Yaskawa INFORM job: OK_R2_O38-47,64(2)(90,0)_MPOK.JBI

/JOB
//NAME OK_R2_O38-47,64(2)(90,0)_MPOK
///FOLDERNAME X4
//POS
///NPOS 359,359,359,19,0,0
///TOOL 0
///POSTYPE PULSE
///PULSE
C00000=-102904,-190754,-108658,-56793,33718,43054
C00001=-112112,-124440,-79629,-37912,40591,30924
C00002=-145621,-43895,-45824,-14341,74181,8322
C00003=-153971,-33006,-36006,-12070,72386,5523
C00004=-154957,-31241,-33389,-11833,71552,5253
C00005=-154957,-31059,-32306,-11871,70990,5309
C00006=-154957,-31147,-32820,-11853,71255,5283
C00007=-152959,-34045,-35008,-12435,71415,5986
C00008=-152821,-33501,-33767,-12507,70963,6084
C00009=-152893,-32341,-33000,-12478,71072,6047
C00010=-153154,-34489,-35846,-12359,71666,5891
C00011=-152546,-38024,-38116,-12561,71351,6144
C00012=-150032,-44426,-43245,-13273,71622,7027
C00013=-145621,-43895,-45824,-14341,74181,8322
C00014=-126188,-124725,-79701,-29915,35046,24780
C00015=-102904,-190754,-108658,-56793,33718,43054
C00016=-131529,-189509,-110128,-36771,24434,27261
C00017=-124211,-86804,-80218,-19393,77786,15538
C00018=-160160,17664,-548,-10057,75687,3034
C00019=-160660,22954,7322,-10002,73531,3037
C00020=-166212,32109,17444,-8387,71396,1231
C00021=-166212,32264,18572,-8416,70786,1274
C00022=-166212,32192,18060,-8403,71061,1255
C00023=-166132,29456,15334,-8416,71338,1265
C00024=-166132,29543,15979,-8433,70989,1289
C00025=-166315,30482,16900,-8379,70890,1229
C00026=-166283,28892,15324,-8381,71043,1230
C00027=-165319,19573,3695,-8574,73487,1399
C00028=-163582,7043,-11027,-8999,76267,1804
C00029=-162101,-9402,-41897,-5301,86162,910
C00030=-133469,39121,-1061,931,85072,6891
C00031=-135751,46408,8355,1655,83056,6142
C00032=-135516,49476,14058,1587,81119,6193
C00033=-135516,49311,14679,1588,80652,6188
C00034=-135036,46950,11602,1434,81323,6352
C00035=-134946,46723,11962,1405,80982,6377
C00036=-135074,47950,13285,1445,80801,6333
C00037=-135102,44394,8734,1452,81774,6335
C00038=-133469,39121,-1061,931,85072,6891
C00039=-135146,16919,-22910,1456,87131,6386
C00040=-160578,-137207,-111137,27103,45167,-7155
C00041=-166532,-153428,-115250,33739,42272,-11545
C00042=-166532,-153428,-115250,33739,42272,-11545
C00043=-160883,-131526,-133102,-3483,78120,-6366
C00044=-103370,-159686,-136025,-1765,64172,-8056
C00045=-97179,-138237,-129333,-10238,76593,11306
C00046=-96065,-128281,-122439,-10507,77596,11607
C00047=-96065,-128106,-120653,-10546,76604,11690
C00048=-96065,-128281,-122439,-10507,77596,11607
C00049=-96974,-121186,-120234,-10189,79734,11117
C00050=-96065,-128281,-122439,-10507,77596,11607
C00051=-80019,-98046,-111669,-14399,88698,15911
C00052=-80077,-97852,-111516,-14385,88694,15892
C00053=-80077,-98331,-110658,-14385,87944,15982
C00054=-80077,-97897,-111441,-14385,88627,15900
C00055=-80867,-94680,-110202,-14197,89359,15553
C00056=-80077,-97897,-111441,-14385,88627,15900
C00057=-77060,-103837,-123440,-15157,93336,16325
C00058=-77104,-103620,-123385,-15148,93404,16303
C00059=-82212,-117279,-126602,-8714,87753,18646
C00060=-83304,-119533,-127995,-7425,87342,19011
C00061=-83304,-120285,-126924,-7427,86307,19072
C00062=-83304,-120125,-127175,-7427,86540,19060
C00063=-84285,-114583,-125380,-7184,88184,18645
C00064=-83304,-120125,-127175,-7427,86540,19060
C00065=-78124,-131037,-133000,-8681,85036,20864
C00066=-78124,-131037,-133000,-8681,85036,20864
C00067=-80781,-132367,-131851,-8063,83392,20088
C00068=-80781,-132658,-130737,-8071,82565,20142
C00069=-80781,-132579,-131090,-8068,82820,20125
C00070=-82215,-124520,-128659,-7695,85306,19491
C00071=-80136,-136061,-133167,-8229,82377,20371
C00072=-80218,-134686,-135534,-8183,84509,20204
C00073=-75563,-118157,-129697,-13391,92336,27261
C00074=-84024,-123631,-127734,-11595,87159,24981
C00075=-84024,-123979,-126960,-11598,86516,25042
C00076=-84024,-123746,-127494,-11596,86956,25000
C00077=-85048,-122093,-126977,-11373,87337,24623
C00078=-81994,-135324,-132084,-12059,84184,25946
C00079=-81994,-133752,-136174,-12028,87438,25630
C00080=-81994,-133752,-136174,-12028,87438,25630
C00081=-83107,-120864,-125937,-11789,87596,25245
C00082=-83880,-119254,-122492,-11630,86222,25116
C00083=-83880,-119583,-121326,-11637,85351,25197
C00084=-83880,-119399,-122020,-11633,85865,25149
C00085=-85062,-113328,-120022,-11369,87556,24598
C00086=-83880,-119399,-122020,-11633,85865,25149
C00087=-83464,-119333,-123502,-11716,86850,25194
C00088=-84085,-116294,-122008,-11580,87393,24935
C00089=-84085,-116863,-120480,-11583,86184,25047
C00090=-84085,-116689,-121008,-11580,86590,25010
C00091=-85140,-111307,-119205,-11348,88071,24523
C00092=-84085,-116194,-122230,-11576,87577,24918
C00093=-82864,-118268,-130611,-11862,91757,24924
C00094=-82864,-118268,-130611,-11862,91757,24924
C00095=-86851,-110557,-120071,-10968,88745,23893
C00096=-86851,-111341,-118540,-10968,87421,24011
C00097=-86851,-110811,-119621,-10968,88345,23929
C00098=-88598,-109546,-119189,-10575,88500,23337
C00099=-86851,-110811,-119621,-10968,88345,23929
C00100=-83825,-124590,-131318,-11630,88867,24881
C00101=-82909,-127853,-136097,-11834,90233,25054
C00102=-84148,-125178,-125504,-11579,85018,25131
C00103=-81186,-118241,-121828,-12198,86718,25964
C00104=-81186,-118533,-120824,-12201,85966,26037
C00105=-81186,-118483,-121017,-12200,86107,26023
C00106=-82314,-113243,-119285,-11952,87535,25506
C00107=-81186,-118241,-121828,-12198,86718,25964
C00108=-87931,-140644,-131144,-10841,80108,24284
C00109=-89960,-139833,-128047,-10433,78377,23732
C00110=-89960,-139550,-127065,-10448,77925,23770
C00111=-89960,-139622,-127307,-10444,78035,23761
C00112=-90753,-134395,-125809,-10209,79670,23349
C00113=-89456,-143397,-129529,-10578,77538,23979
C00114=-95203,-107502,-133483,-6717,98684,21003
C00115=-95203,-107502,-133483,-6717,98684,21003
C00116=70091,-137861,-134613,19540,89589,-11549
C00117=70091,-137861,-134613,19540,89589,-11549
C00118=89914,-142582,-130695,14485,81723,-10120
C00119=90202,-137048,-128128,14398,82897,-9883
C00120=90202,-136718,-126391,14423,82025,-9985
C00121=90202,-136862,-127082,14413,82365,-9945
C00122=91010,-131454,-125503,14223,83978,-9478
C00123=90202,-137070,-128271,14397,82970,-9874
C00124=76195,-137070,-128271,14397,82970,-9874
C00125=74994,-123934,-123423,14560,86840,-9835
C00126=74994,-124092,-122198,14564,86029,-9931
C00127=74994,-124005,-122955,14561,86525,-9872
C00128=76141,-119465,-121513,14342,87728,-9340
C00129=72631,-133219,-128550,14998,85696,-10781
C00130=72631,-131663,-134232,14989,89852,-10278
C00131=50716,-132590,-134806,14983,95067,-21778
C00132=53786,-122460,-125023,14607,93736,-20890
C00133=54881,-121663,-124068,14472,93371,-20558
C00134=54881,-122014,-122728,14450,92397,-20672
C00135=54881,-121856,-123398,14460,92875,-20616
C00136=56721,-117465,-121986,14267,93906,-19868
C00137=54881,-121856,-123398,14460,92875,-20616
C00138=55322,-120745,-123309,14420,93300,-20415
C00139=55322,-120747,-123302,14420,93295,-20416
C00140=55322,-120978,-122461,14407,92679,-20487
C00141=55322,-120864,-122902,14414,92999,-20450
C00142=56710,-117554,-121835,14266,93775,-19889
C00143=54436,-122887,-123768,14509,92662,-20793
C00144=54436,-122067,-126198,14556,94519,-20574
C00145=53688,-126302,-127242,14482,93230,-21000
C00146=7968,-117738,-135568,14910,102458,-19890
C00147=7968,-117738,-135568,14910,102458,-19890
C00148=4119,-116606,-125698,15061,97809,-21757
C00149=7770,-114903,-122318,14590,96007,-20739
C00150=7770,-115418,-121244,14557,95111,-20843
C00151=7770,-115024,-122084,14598,95810,-20761
C00152=9375,-110655,-120613,14452,96836,-20097
C00153=7770,-115024,-122084,14598,95810,-20761
C00154=10569,-102485,-118509,17167,107955,-30726
C00155=17008,-101176,-116544,17116,107524,-30934
C00156=-121481,-92648,-105286,-5369,115019,-86755
C00157=-120615,-96829,-107734,-5213,114434,-86412
C00158=23859,-150611,-131722,11614,81196,-13147
C00159=5605,-98558,-114313,9016,91646,-19053
C00160=5292,-97369,-113802,9089,91971,-19129
C00161=5881,-109040,-123705,8960,92007,-18939
C00162=6434,-120006,-133010,8839,92040,-18760
C00163=-12667,-120051,-129788,-19636,91452,63850
C00164=-15640,-171133,-136982,-20070,70138,66271
C00165=3779,-163113,-125940,-36463,74354,73480
C00166=-120436,-95190,-80290,-14692,43277,16053
C00167=-119715,-95468,-78930,-15521,42464,16563
C00168=1349,-140937,-118482,-38247,78517,71026
C00169=-15636,-141614,-117585,-35447,65083,67762
C00170=-17609,-126505,-112505,-34601,67163,66072
C00171=-24043,-118481,-124771,-21586,79008,61529
C00172=-24043,-118481,-124771,-21586,79008,61529
C00173=-75030,-118005,-124618,-21594,79160,61521
C00174=-115715,-153549,-128562,15788,54400,49074
C00175=-122131,-153692,-122292,24372,49463,44977
C00176=-120438,-96789,-101713,-1489,48968,3516
C00177=-120356,-99154,-104149,-1548,49253,3547
C00178=-84198,-116806,-111213,1772,54897,61304
C00179=-87160,-120534,-109364,10018,48087,58269
C00180=-90828,-138253,-118809,13315,45388,56216
C00181=-90828,-138253,-118809,13315,45388,56216
C00182=-90828,-142934,-129815,12421,49655,56806
C00183=-90829,-142933,-129813,12421,49658,56806
C00184=-119872,-163920,-132846,33283,49576,42941
C00185=-126991,-146326,-124104,35016,55490,41598
C00186=-120835,-94912,-106201,4597,84031,3620
C00187=-120296,-100536,-106811,4468,81494,3706
C00188=-119922,-143587,-123205,31413,53438,44308
C00189=-77415,-98459,-105381,5383,51560,63214
C00190=-71925,-92447,-101662,533,50488,65336
C00191=-77718,-122737,-116129,5642,44048,62545
C00192=-53268,-154266,-130714,-22807,48565,72872
C00193=-53268,-154266,-130714,-22807,48565,72872
C00194=-65704,-162398,-123942,-17029,37659,69009
C00195=-69631,-160797,-117543,-19584,31037,68677
C00196=-120621,-91661,-79831,4809,93096,-80691
C00197=-120610,-95504,-82099,4805,92519,-80709
C00198=-64928,-151300,-115352,-22074,35531,70301
C00199=-55359,-110208,-106429,-19631,55099,70468
C00200=-56474,-111761,-106561,-17625,52293,70865
C00201=-58794,-112885,-105581,-13565,47681,71177
C00202=-50265,-141050,-116073,-27906,38980,77613
C00203=-41790,-175398,-134696,-41509,59591,72504
C00204=-40096,-167295,-132799,-40833,62675,71982
C00205=-66805,-175580,-133819,-17842,44997,58057
C00206=-120613,-98309,-97516,-18774,58387,20033
C00207=-120296,-100165,-96633,-19249,57041,20409
C00208=-66730,-175408,-133780,-17867,45074,58078
C00209=-65136,-170814,-132569,-18309,46965,58464
C00210=-52364,-139651,-124628,-28315,65404,66743
C00211=-50532,-107164,-114440,-27328,75285,64992
C00212=-50521,-107002,-114383,-27326,75331,64985
C00213=-56147,-114427,-116211,-21096,65709,65656
C00214=-54523,-105936,-113271,-21470,68505,65739
C00215=-49750,-132075,-132074,-23871,68057,67633
C00216=-51888,-141517,-135531,-28423,71943,65142
C00217=-58410,-142164,-121837,-32385,67064,69630
C00218=-58892,-132878,-117266,-33819,71370,71170
C00219=-120621,-92022,-79948,-5717,93324,-87803
C00220=-120611,-95871,-82213,-5711,92744,-87773
C00221=-91898,-177824,-128316,2778,37745,41927
C00222=-76561,-127099,-115440,3526,55962,41360
C00223=-98908,-102884,-107387,29228,75304,22104
C00224=-100715,-115554,-120696,29641,77391,21955
C00225=-99511,-125054,-130815,29118,78165,22610
C00226=30978,-142903,-136378,16839,87530,-25088
C00227=48053,-137432,-126920,10736,83825,-19877
C00228=-120514,-92773,-72492,63824,26217,-40707
C00229=-122096,-91517,-72885,63277,27653,-40461
C00230=46723,-132150,-125263,10235,84639,-20316
C00231=38144,-96146,-111322,6693,87070,-23612
C00232=36690,-89699,-108774,7082,88920,-23976
C00233=38688,-150385,-135608,6755,74185,-24124
C00234=34744,-121097,-133452,9828,92546,-23976
C00235=92930,-150385,-135608,6755,74185,-24124
C00236=107101,-138400,-125652,2740,73384,-19202
C00237=-120610,-93305,-77258,53115,31058,22991
C00238=-120294,-94166,-75974,54567,30127,22239
C00239=116035,-135916,-124846,-7405,75208,-6894
C00240=75429,-100276,-113037,4073,85400,-20589
C00241=88876,-89136,-108695,-11365,90939,-2676
C00242=92139,-118134,-128268,-12138,88585,-1394
C00243=96790,-150711,-134355,-17072,70659,2161
C00244=96790,-150711,-134355,-17072,70659,2161
C00245=652,-114254,-134536,-4800,91191,-3391
C00246=-166532,-153428,-115250,33739,42272,-11545
C00247=-166532,-153428,-115250,33739,42272,-11545
C00248=-124114,-84683,-61597,-48557,28871,-52530
C00249=-120672,9825,17632,-53753,29009,-53309
C00250=-120673,9828,17635,-53752,29009,-53309
C00251=-119969,9889,17391,-53999,29527,-53154
C00252=-120673,10502,19535,-54974,28515,-52685
C00253=-120213,7916,15945,-54003,29309,-53162
C00254=-120673,9268,16917,-53528,29103,-53422
C00255=-120673,9346,17029,-53570,29085,-53403
C00256=-120325,9631,17167,-53735,29324,-53303
C00257=-120673,9869,17671,-53754,29008,-53308
C00258=-120672,9864,17667,-53755,29008,-53308
C00259=-124114,-84683,-61597,-48557,28871,-52530
C00260=-131339,-154294,-79414,-109628,16862,-24377
C00261=-234701,-24447,-54419,57638,71697,57534
C00262=-192045,-4471,-49137,31395,56880,70337
C00263=-172212,48807,-7818,-1281,85806,67502
C00264=-182022,60397,16725,362,120111,76099
C00265=-181268,75249,48221,-1582,120068,76073
C00266=-181077,73835,47696,-1507,119669,76155
C00267=-181356,72617,44998,-1625,120698,76029
C00268=-181183,75410,49585,-1539,119314,76118
C00269=-180483,73010,46710,-1298,119861,76386
C00270=-180498,74390,47192,-1310,120274,76376
C00271=-180299,81057,52347,-1242,120531,76452
C00272=-174789,63735,852,-597,96026,66536
C00273=-179792,32070,-16354,13350,79915,65662
C00274=-186878,-39073,-38836,41246,34970,63358
C00275=-187481,-32249,-33448,41583,35400,63192
C00276=-188256,-32514,-32154,43117,35074,62369
C00277=-188651,-34827,-34931,42941,35654,62475
C00278=-186711,-32763,-33884,40918,35040,63531
C00279=-187464,-35744,-36703,41375,35550,63305
C00280=-188726,-40923,-42933,41373,37038,63352
C00281=-196569,5763,-30645,36969,53415,67065
C00282=-234701,-24447,-54419,57638,71697,57534
C00283=-149956,-143190,-113193,-9671,18752,-75469
C00284=-134160,-28568,-62536,-18892,48395,-71822
C00285=-120672,9794,17604,-61241,37188,-52240
C00286=-120672,9794,17604,-61241,37188,-52240
C00287=-120555,9400,17043,-61125,37334,-52300
C00288=-120673,9158,15746,-60306,37604,-52768
C00289=-120213,7880,15913,-61361,37506,-52152
C00290=-120673,9106,16782,-61064,37264,-52340
C00291=-120673,9123,16797,-61065,37265,-52339
C00292=-120025,10235,17860,-61424,37632,-52107
C00293=-120673,9754,17568,-61239,37189,-52241
C00294=-120672,9754,17569,-61239,37189,-52241
C00295=-134138,-28506,-62498,-18910,48408,-71815
C00296=-154186,-159927,-117173,-847,12331,-79725
C00297=-85861,-99082,-105113,-44329,59147,-50836
C00298=-83984,-106882,-107996,-46165,58479,-49488
C00299=-120674,-14372,-36148,-15341,86455,-69375
C00300=-120676,-10921,-33498,-15340,86592,-69392
C00301=-120766,11309,-16496,-15719,100731,-71202
C00302=-121175,-12454,-34682,-15229,86445,-69544
C00303=-120675,-14159,-37235,-15335,87207,-69469
C00304=-122749,15787,-12070,-15993,104016,-72342
C00305=-120676,-11639,-34054,-15340,86566,-69391
C00306=-120674,-14390,-36162,-15341,86455,-69375
C00307=-120676,-14354,-36134,-15765,85734,14225
C00308=-120676,-14354,-36134,-15765,85734,14225
C00309=-120809,-13585,-35576,-15734,85761,14174
C00310=-120676,-14158,-37234,-15757,86484,14129
C00311=-120165,-16255,-37568,-15883,85739,14397
C00312=-123124,-16243,-37493,-15196,85151,13465
C00313=-120676,-14374,-36149,-15765,85733,14224
C00314=-120676,-14373,-36148,-15765,85733,14225
C00315=-98406,-95981,-107671,-30899,65126,25478
C00316=-97498,-103141,-110365,-31836,63713,26282
C00317=-158741,-152165,-85078,-53213,16407,-64133
C00318=-151185,-64492,-56891,-27025,41971,-76525
C00319=-187574,37417,13419,2960,77279,72462
C00320=-187020,38831,14880,2796,77088,72647
C00321=-180715,58337,34412,-9745,85564,73616
C00322=-187315,39588,15664,2886,77004,72543
C00323=-187570,37474,12233,2951,78037,72481
C00324=-180247,63606,40673,-12018,86600,73536
C00325=-187574,37421,13424,2960,77279,72462
C00326=-187576,37412,13414,2961,77280,72461
C00327=-187610,37331,13331,3255,76507,-7692
C00328=-182719,57686,35499,-3659,79600,-3173
C00329=-182518,60502,39600,-3732,78534,-3072
C00330=-187825,35310,11263,3318,76749,-7758
C00331=-187564,37491,12251,3232,77251,-7657
C00332=-186627,65968,46003,-2806,77236,-4449
C00333=-187574,37420,13423,3244,76495,-7680
C00334=-174916,2091,-20307,-7000,70210,-31977
C00335=-151185,-64492,-56891,-27025,41971,-76525
C00336=-158741,-152165,-85078,-53213,16407,-64133
C00337=-136335,-97157,-88666,-6240,65884,-69249
C00338=-141826,-62430,-72987,-3929,73707,-71532
C00339=-140052,-21130,-52867,24635,78479,-75610
C00340=-137473,58120,11150,19511,106253,-71077
C00341=-132799,89049,47439,16428,114143,-68872
C00342=-132090,97611,56676,15970,118552,-68089
C00343=-132116,97401,56917,15786,119997,-67945
C00344=-135984,107314,69748,14048,119719,-69614
C00345=-135785,103774,66356,14147,119946,-69504
C00346=-131685,106105,70627,22443,116548,-67586
C00347=-133954,98465,50155,16232,124944,-67916
C00348=-142400,32764,-15276,22713,92529,-74169
C00349=-109290,70352,15308,-18647,88059,-61302
C00350=-83699,85527,52785,-52979,68456,-51263
C00351=-80420,18251,15496,-64356,57036,-45994
C00352=-80421,18253,15498,-64356,57035,-45994
C00353=-80264,19576,16606,-64391,57138,-45967
C00354=-80421,18695,17178,-64825,56670,-45601
C00355=-79680,17143,14466,-64475,57547,-45892
C00356=-77796,32158,28786,-65456,58289,-45032
C00357=-78671,21218,15982,-64051,58734,-46270
C00358=-89230,-40025,-45988,-57168,55507,-51535
BC00000=155275,760074,251743
BC00001=155275,819591,251743
BC00002=155275,819591,251743
BC00003=155275,819591,251743
BC00004=155275,819591,251743
BC00005=155275,819591,251743
BC00006=155275,819591,251743
BC00007=155275,819591,251743
BC00008=155275,819591,251743
BC00009=155275,819591,251743
BC00010=155275,819591,251743
BC00011=155275,819591,251743
BC00012=155275,819591,251743
BC00013=155275,819591,251743
BC00014=155275,819591,251743
BC00015=155275,760074,251743
BC00016=334637,762746,239047
BC00017=334637,842186,239047
BC00018=334637,842186,239047
BC00019=334637,842186,239047
BC00020=334637,842186,239047
BC00021=334637,842186,239047
BC00022=334637,842186,239047
BC00023=334637,842186,239047
BC00024=334637,842186,239047
BC00025=334637,842186,239047
BC00026=334637,842186,239047
BC00027=334637,842186,239047
BC00028=334637,842186,239047
BC00029=336476,842187,209320
BC00030=343292,842193,99157
BC00031=343292,842193,99157
BC00032=343292,842193,99157
BC00033=343292,842193,99157
BC00034=343292,842193,99157
BC00035=343292,842193,99157
BC00036=343292,842193,99157
BC00037=343292,842193,99157
BC00038=343292,842193,99157
BC00039=343292,842193,99157
BC00040=343292,842193,99157
BC00041=343292,714597,99157
BC00042=343292,714597,1074810
BC00043=343292,714597,1074810
BC00044=343292,942381,1074810
BC00045=336034,956109,1074810
BC00046=336034,956109,1074810
BC00047=336034,956109,1074810
BC00048=336034,956109,1074810
BC00049=336034,956109,1074810
BC00050=336034,956109,1074810
BC00051=336034,956109,1074810
BC00052=336034,956109,1074810
BC00053=336034,956109,1074810
BC00054=336034,956109,1074810
BC00055=336034,956109,1074810
BC00056=336034,956109,1074810
BC00057=336034,956109,1074810
BC00058=371500,1003655,1072368
BC00059=371500,1011303,1072368
BC00060=371500,1012871,1072368
BC00061=371500,1012871,1072368
BC00062=371500,1012871,1072368
BC00063=371500,1012871,1072368
BC00064=371500,1012871,1072368
BC00065=371500,1012871,1072368
BC00066=310141,1007143,1071829
BC00067=310141,1007143,1071829
BC00068=310141,1007143,1071829
BC00069=310141,1007143,1071829
BC00070=310141,1007143,1071829
BC00071=310141,1007143,1071829
BC00072=310141,1007143,1071829
BC00073=246928,976807,1071829
BC00074=246928,976807,1071829
BC00075=246928,976807,1071829
BC00076=246928,976807,1071829
BC00077=246928,976807,1071829
BC00078=246928,976807,1071829
BC00079=246928,976807,1071829
BC00080=144012,964080,1063254
BC00081=144012,964080,1063254
BC00082=144012,964080,1063254
BC00083=144012,964080,1063254
BC00084=144012,964080,1063254
BC00085=144012,964080,1063254
BC00086=144012,964080,1063254
BC00087=107418,957008,1063254
BC00088=107418,957008,1063254
BC00089=107418,957008,1063254
BC00090=107418,957008,1063254
BC00091=107418,957008,1063254
BC00092=107418,957008,1063254
BC00093=107418,957008,1063254
BC00094=126016,899142,1063254
BC00095=126016,899142,1063254
BC00096=126016,899142,1063254
BC00097=126016,899142,1063254
BC00098=126016,899142,1063254
BC00099=126016,899142,1063254
BC00100=126016,899142,1063254
BC00101=32383,899142,1063254
BC00102=33723,949074,1063254
BC00103=33723,949074,1063254
BC00104=33723,949074,1063254
BC00105=33723,949074,1063254
BC00106=33723,949074,1063254
BC00107=33723,949074,1063254
BC00108=7047,944370,1063254
BC00109=6971,946386,1064283
BC00110=6971,946386,1064283
BC00111=6971,946386,1064283
BC00112=6971,946386,1064283
BC00113=6971,946386,1064283
BC00114=6971,946386,1064283
BC00115=25103,830564,1064283
BC00116=1840,976824,1064283
BC00117=1840,1022624,1064283
BC00118=1840,1022624,1064283
BC00119=1840,1022624,1064283
BC00120=1840,1022624,1064283
BC00121=1840,1022624,1064283
BC00122=1840,1022624,1064283
BC00123=1840,1022624,1064283
BC00124=32240,1021120,1065802
BC00125=32240,1021120,1065802
BC00126=32240,1021120,1065802
BC00127=32240,1021120,1065802
BC00128=32240,1021120,1065802
BC00129=32240,1021120,1065802
BC00130=32240,1021120,1065802
BC00131=75978,1001728,1065802
BC00132=75977,1001729,1065799
BC00133=75977,1001729,1065799
BC00134=75977,1001729,1065799
BC00135=75977,1001729,1065799
BC00136=75977,1001729,1065799
BC00137=75977,1001729,1065799
BC00138=117549,1001729,1065799
BC00139=117549,1001729,1065799
BC00140=117549,1001729,1065799
BC00141=117549,1001729,1065799
BC00142=117549,1001729,1065799
BC00143=117549,1001729,1065799
BC00144=117549,1001729,1065799
BC00145=56674,1036312,1065895
BC00146=56674,1036312,1065895
BC00147=30889,1102979,1065895
BC00148=45214,1102979,1065895
BC00149=45214,1102979,1065895
BC00150=45214,1102979,1065895
BC00151=45214,1102978,1065892
BC00152=45214,1102978,1065892
BC00153=45214,1102978,1065892
BC00154=45214,1102978,1065889
BC00155=45214,1102978,1065889
BC00156=145257,917701,1075175
BC00157=145257,917701,1075175
BC00158=45214,1102978,1065887
BC00159=45214,1102978,1065887
BC00160=45214,1102978,1065887
BC00161=45214,1102978,1065887
BC00162=45214,1102978,1065887
BC00163=50349,952936,1065887
BC00164=50349,952936,1065887
BC00165=50349,952936,1065887
BC00166=156935,778985,1075175
BC00167=156935,778985,1075175
BC00168=50349,952936,1065887
BC00169=72136,952936,1065887
BC00170=72136,952936,1065887
BC00171=72136,952936,1065887
BC00172=58646,939592,1065887
BC00173=33,880302,1065887
BC00174=33,928742,1065885
BC00175=33,928742,1065885
BC00176=369319,873480,1075175
BC00177=369319,873480,1075175
BC00178=33,928742,1065885
BC00179=33,928742,1065885
BC00180=33,928742,1065885
BC00181=33,926822,1072255
BC00182=33,849370,1070063
BC00183=271563,976879,1070062
BC00184=312671,982863,1065015
BC00185=312671,982863,1065015
BC00186=4086,859403,1075175
BC00187=4086,859403,1075175
BC00188=312671,982863,1065015
BC00189=312671,982863,1065015
BC00190=312671,982863,1065015
BC00191=312671,982863,1065015
BC00192=312671,982863,1065015
BC00193=280596,959851,1065015
BC00194=280596,959851,1065015
BC00195=280596,959851,1065015
BC00196=125992,771300,1075175
BC00197=125992,771300,1075175
BC00198=280596,959851,1065015
BC00199=280596,959851,1065012
BC00200=280596,959851,1065013
BC00201=280596,959851,1065015
BC00202=280596,959851,1065015
BC00203=280596,959851,1065015
BC00204=211687,973675,1065015
BC00205=204246,973675,1065015
BC00206=168833,851602,1075175
BC00207=168833,851602,1075175
BC00208=204246,973675,1065015
BC00209=204246,973675,1065015
BC00210=204246,973675,1065015
BC00211=204246,973675,1065015
BC00212=204246,973675,1065015
BC00213=204246,973675,1065015
BC00214=204246,973675,1065015
BC00215=204246,973675,1065015
BC00216=93803,958451,1065015
BC00217=93803,958451,1065015
BC00218=93804,958451,1065014
BC00219=27668,771045,1075175
BC00220=27668,771045,1075175
BC00221=93804,958451,1065014
BC00222=93804,958451,1065014
BC00223=93804,958451,1065014
BC00224=93804,958451,1065014
BC00225=93804,958451,1065014
BC00226=58899,987526,1068118
BC00227=58899,987526,1068118
BC00228=345503,839022,1075175
BC00229=345503,839022,1075175
BC00230=58899,987526,1068118
BC00231=58899,987526,1068118
BC00232=58899,987526,1068118
BC00233=58899,987526,1068118
BC00234=58139,987526,1068216
BC00235=1984,1028862,1068118
BC00236=1984,1028862,1068118
BC00237=310150,835828,1075175
BC00238=310150,835828,1075175
BC00239=1984,1028862,1068118
BC00240=1984,1028862,1068118
BC00241=1984,1028862,1068118
BC00242=1984,1028862,1068118
BC00243=1984,1028862,1068118
BC00244=1984,833796,1068118
BC00245=56336,759226,1064779
BC00246=343292,714597,1074810
BC00247=343292,714597,99157
BC00248=326718,829986,221879
BC00249=326019,834851,227054
BC00250=323796,839870,208138
BC00251=322906,841877,200572
BC00252=322906,841877,200572
BC00253=322906,841877,200572
BC00254=327037,844194,200572
BC00255=331719,846821,200572
BC00256=335850,849138,200572
BC00257=336739,847130,208139
BC00258=338963,842112,227055
BC00259=326718,829986,221879
BC00260=326718,721817,221879
BC00261=301908,735078,53
BC00262=301908,735078,53
BC00263=257340,761494,53
BC00264=218510,827652,130053
BC00265=218510,827652,130053
BC00266=218510,827652,130053
BC00267=218510,827652,130053
BC00268=218510,827652,130053
BC00269=218510,827652,130053
BC00270=218510,827652,130053
BC00271=218510,827652,130053
BC00272=257340,761494,53
BC00273=243122,776164,27952
BC00274=213981,806232,85133
BC00275=213981,806232,85133
BC00276=213981,806232,85133
BC00277=213981,806232,85133
BC00278=213981,806232,85133
BC00279=213981,806232,85133
BC00280=213981,806232,85133
BC00281=301908,735078,53
BC00282=301908,735078,53
BC00283=326019,716112,4997
BC00284=326019,754467,4997
BC00285=315535,829024,226895
BC00286=312111,833369,207979
BC00287=310742,835107,200413
BC00288=310742,835107,200413
BC00289=310742,835107,200413
BC00290=306612,832790,200413
BC00291=301791,830087,200413
BC00292=297661,827770,200413
BC00293=299030,826032,207979
BC00294=302454,821686,226895
BC00295=326019,802314,4997
BC00296=326019,740906,5323
BC00297=131939,688818,32608
BC00298=131939,774315,32608
BC00299=131939,801396,210359
BC00300=131334,801067,183577
BC00301=131093,800936,172865
BC00302=131093,800936,172865
BC00303=131093,800936,172865
BC00304=131093,800936,172865
BC00305=125276,797669,183577
BC00306=125880,797998,210358
BC00307=132304,800008,176562
BC00308=128880,804353,157646
BC00309=127511,806091,150080
BC00310=127511,806091,150080
BC00311=127511,806091,150080
BC00312=127511,806091,150080
BC00313=122408,800723,157646
BC00314=125832,796378,176562
BC00315=132304,777362,53
BC00316=132304,687429,53
BC00317=341619,775319,231168
BC00318=341619,843929,231168
BC00319=341619,843929,231168
BC00320=341015,843600,204386
BC00321=340773,843469,193674
BC00322=340773,843469,193674
BC00323=340773,843469,193674
BC00324=340773,843469,193674
BC00325=338609,842251,204386
BC00326=339214,842580,231168
BC00327=349631,842380,197374
BC00328=349631,842380,197374
BC00329=349631,842380,197374
BC00330=344838,853004,170892
BC00331=344838,853004,170892
BC00332=349631,842380,197374
BC00333=336550,839583,197374
BC00334=338313,841095,209130
BC00335=341619,843929,231168
BC00336=341619,775319,231168
BC00337=190901,728772,170929
BC00338=190901,786037,170929
BC00339=193011,793039,131574
BC00340=182032,791881,61669
BC00341=176016,791246,23364
BC00342=175802,792372,8727
BC00343=178212,792700,4465
BC00344=193011,793039,53
BC00345=193011,793039,53
BC00346=178212,792700,4465
BC00347=178845,792714,4276
BC00348=193612,789752,91438
BC00349=126346,753501,53
BC00350=70335,723316,53
BC00351=93918,779758,165352
BC00352=91695,784776,146437
BC00353=90805,786784,138870
BC00354=90805,786784,138870
BC00355=90805,786784,138870
BC00356=90805,786784,138870
BC00357=90805,786784,138870
BC00358=106862,787018,165353
EC00000=798156,0
EC00001=798156,0
EC00002=798156,0
EC00003=798156,0
EC00004=798156,0
EC00005=798156,0
EC00006=798156,0
EC00007=798156,0
EC00008=798156,0
EC00009=798156,0
EC00010=798156,0
EC00011=798156,0
EC00012=798156,0
EC00013=798156,0
EC00014=798156,0
EC00015=798156,0
EC00016=798156,0
EC00017=798156,0
EC00018=798156,0
EC00019=798156,0
EC00020=798156,0
EC00021=798156,0
EC00022=798156,0
EC00023=798156,0
EC00024=798156,0
EC00025=798156,0
EC00026=798156,0
EC00027=798156,0
EC00028=798156,0
EC00029=798156,0
EC00030=798156,0
EC00031=798156,0
EC00032=798156,0
EC00033=798156,0
EC00034=798156,0
EC00035=798156,0
EC00036=798156,0
EC00037=798156,0
EC00038=798156,0
EC00039=798156,0
EC00040=798156,0
EC00041=798156,0
EC00042=798156,0
EC00043=798156,0
EC00044=798156,0
EC00045=798156,0
EC00046=798156,0
EC00047=798156,0
EC00048=798156,0
EC00049=798156,0
EC00050=798156,0
EC00051=798156,0
EC00052=798156,0
EC00053=798156,0
EC00054=798156,0
EC00055=798156,0
EC00056=798156,0
EC00057=798156,0
EC00058=798156,0
EC00059=798156,0
EC00060=798156,0
EC00061=798156,0
EC00062=798156,0
EC00063=798156,0
EC00064=798156,0
EC00065=798156,0
EC00066=798156,0
EC00067=798156,0
EC00068=798156,0
EC00069=798156,0
EC00070=798156,0
EC00071=798156,0
EC00072=798156,0
EC00073=798156,0
EC00074=798156,0
EC00075=798156,0
EC00076=798156,0
EC00077=798156,0
EC00078=798156,0
EC00079=798156,0
EC00080=798156,0
EC00081=798156,0
EC00082=798156,0
EC00083=798156,0
EC00084=798156,0
EC00085=798156,0
EC00086=798156,0
EC00087=798156,0
EC00088=798156,0
EC00089=798156,0
EC00090=798156,0
EC00091=798156,0
EC00092=798156,0
EC00093=798156,0
EC00094=798156,0
EC00095=798156,0
EC00096=798156,0
EC00097=798156,0
EC00098=798156,0
EC00099=798156,0
EC00100=798156,0
EC00101=798156,0
EC00102=798156,0
EC00103=798156,0
EC00104=798156,0
EC00105=798156,0
EC00106=798156,0
EC00107=798156,0
EC00108=798156,0
EC00109=798156,0
EC00110=798156,0
EC00111=798156,0
EC00112=798156,0
EC00113=798156,0
EC00114=798156,0
EC00115=798156,0
EC00116=798156,0
EC00117=798156,0
EC00118=798156,0
EC00119=798156,0
EC00120=798156,0
EC00121=798156,0
EC00122=798156,0
EC00123=798156,0
EC00124=798156,0
EC00125=798156,0
EC00126=798156,0
EC00127=798156,0
EC00128=798156,0
EC00129=798156,0
EC00130=798156,0
EC00131=798156,0
EC00132=798154,0
EC00133=798154,0
EC00134=798154,0
EC00135=798154,0
EC00136=798154,0
EC00137=798154,0
EC00138=798154,0
EC00139=798154,0
EC00140=798154,0
EC00141=798154,0
EC00142=798154,0
EC00143=798154,0
EC00144=798154,0
EC00145=799965,0
EC00146=799965,0
EC00147=799965,0
EC00148=799965,0
EC00149=799965,0
EC00150=799965,0
EC00151=799962,1
EC00152=799962,1
EC00153=799962,1
EC00154=799960,2
EC00155=799960,2
EC00156=975524,0
EC00157=975524,0
EC00158=799958,2
EC00159=799958,2
EC00160=799958,2
EC00161=799958,2
EC00162=799958,2
EC00163=799958,2
EC00164=799958,2
EC00165=799958,2
EC00166=975524,0
EC00167=975524,0
EC00168=799958,2
EC00169=799958,2
EC00170=799958,2
EC00171=799958,2
EC00172=799958,2
EC00173=799958,2
EC00174=799955,2
EC00175=799955,2
EC00176=975524,0
EC00177=975524,0
EC00178=799955,2
EC00179=799955,2
EC00180=799955,2
EC00181=799955,2
EC00182=799954,3
EC00183=799951,3
EC00184=799951,3
EC00185=799951,3
EC00186=975524,0
EC00187=975524,0
EC00188=799951,3
EC00189=799951,3
EC00190=799951,3
EC00191=799951,3
EC00192=799951,3
EC00193=799951,3
EC00194=799951,3
EC00195=799951,3
EC00196=975524,0
EC00197=975524,0
EC00198=799951,3
EC00199=799949,4
EC00200=799950,4
EC00201=799951,3
EC00202=799951,3
EC00203=799951,3
EC00204=799951,3
EC00205=799951,3
EC00206=975524,0
EC00207=975524,0
EC00208=799951,3
EC00209=799951,3
EC00210=799951,3
EC00211=799951,3
EC00212=799951,3
EC00213=799951,3
EC00214=799951,3
EC00215=799951,3
EC00216=799951,3
EC00217=799951,3
EC00218=799949,3
EC00219=975524,0
EC00220=975524,0
EC00221=799949,3
EC00222=799949,3
EC00223=799949,3
EC00224=799949,3
EC00225=799949,3
EC00226=799949,3
EC00227=799949,3
EC00228=975524,0
EC00229=975524,0
EC00230=799949,3
EC00231=799949,3
EC00232=799949,3
EC00233=799949,3
EC00234=799949,3
EC00235=799949,3
EC00236=799949,3
EC00237=975524,0
EC00238=975524,0
EC00239=799949,3
EC00240=799949,3
EC00241=799949,3
EC00242=799949,3
EC00243=799949,3
EC00244=799949,3
EC00245=802129,3
EC00246=798156,0
EC00247=798156,0
EC00248=798156,0
EC00249=798156,0
EC00250=798156,0
EC00251=798156,0
EC00252=798156,0
EC00253=798156,0
EC00254=798156,0
EC00255=798156,0
EC00256=798156,0
EC00257=798156,0
EC00258=798156,0
EC00259=798156,0
EC00260=798156,0
EC00261=798156,0
EC00262=798156,0
EC00263=798156,0
EC00264=798156,0
EC00265=798156,0
EC00266=798156,0
EC00267=798156,0
EC00268=798156,0
EC00269=798156,0
EC00270=798156,0
EC00271=798156,0
EC00272=798156,0
EC00273=798156,0
EC00274=798156,0
EC00275=798156,0
EC00276=798156,0
EC00277=798156,0
EC00278=798156,0
EC00279=798156,0
EC00280=798156,0
EC00281=798156,0
EC00282=798156,0
EC00283=798156,0
EC00284=798156,0
EC00285=798156,0
EC00286=798156,0
EC00287=798156,0
EC00288=798156,0
EC00289=798156,0
EC00290=798156,0
EC00291=798156,0
EC00292=798156,0
EC00293=798156,0
EC00294=798156,0
EC00295=798156,0
EC00296=798156,0
EC00297=798156,0
EC00298=798156,0
EC00299=798156,0
EC00300=798156,0
EC00301=798156,0
EC00302=798156,0
EC00303=798156,0
EC00304=798156,0
EC00305=798156,0
EC00306=798156,0
EC00307=798156,0
EC00308=798156,0
EC00309=798156,0
EC00310=798156,0
EC00311=798156,0
EC00312=798156,0
EC00313=798156,0
EC00314=798156,0
EC00315=798156,0
EC00316=798156,0
EC00317=798156,0
EC00318=798156,0
EC00319=798156,0
EC00320=798156,0
EC00321=798156,0
EC00322=798156,0
EC00323=798156,0
EC00324=798156,0
EC00325=798156,0
EC00326=798156,0
EC00327=798156,0
EC00328=798156,0
EC00329=798155,1
EC00330=798156,0
EC00331=798156,0
EC00332=798156,0
EC00333=798156,0
EC00334=798156,0
EC00335=798156,0
EC00336=798156,0
EC00337=798156,0
EC00338=798156,0
EC00339=798156,0
EC00340=798156,0
EC00341=798156,0
EC00342=798156,0
EC00343=798156,0
EC00344=798156,0
EC00345=798156,0
EC00346=798156,0
EC00347=798156,0
EC00348=798156,0
EC00349=798156,0
EC00350=798156,0
EC00351=798156,0
EC00352=798156,0
EC00353=798156,0
EC00354=798156,0
EC00355=798156,0
EC00356=798156,0
EC00357=798156,0
EC00358=798156,0
///POSTYPE BASE
///RECTAN
///RCONF 0,0,0,0,0,0,0,0,0,0,0,0,0,0,0,0,0,0,0,0,0,0,0,0
P00006=0.222,-3.123,-1.508,0.0000,0.0000,0.0000
P00021=-0.225,-6.128,-0.405,0.0000,0.0000,0.0000
P00022=0.222,-3.123,-1.508,0.0000,0.0000,0.0000
P00023=0.143,-0.036,0.682,0.0000,0.0000,0.0000
P00030=5.926,-4.294,-1.390,0.0000,0.0000,0.0000
P00031=1.853,-0.001,-1.549,0.0000,0.0000,0.0000
P00032=1.957,0.503,-7.217,0.0000,0.0000,0.0000
///RCONF 0,0,0,0,1,0,0,0,0,0,0,0,0,0,0,0,0,0,0,0,0,0,0,0
P00033=-0.123,0.612,-5.012,0.0000,0.0000,0.0000
///RCONF 0,0,0,0,0,0,0,0,0,0,0,0,0,0,0,0,0,0,0,0,0,0,0,0
P00034=-0.304,0.773,-2.693,0.0000,0.0000,0.0000
P00035=2.817,0.591,-1.622,0.0000,0.0000,0.0000
P00036=-1.108,-0.829,1.850,0.0000,0.0000,0.0000
P00037=0.023,0.937,-2.677,0.0000,0.0000,0.0000
P00038=0.158,-1.133,-1.952,0.0000,0.0000,0.0000
P00039=0.012,-3.081,-0.106,0.0000,0.0000,0.0000
P00040=-0.030,9.648,2.467,0.0000,0.0000,0.0000
P00041=0.192,3.924,0.305,0.0000,0.0000,0.0000
P00042=-0.217,1.941,0.413,0.0000,0.0000,0.0000
P00043=-0.044,-1.937,1.197,0.0000,0.0000,0.0000
P00044=0.687,-2.322,1.156,0.0000,0.0000,0.0000
//INST
///DATE 2025/03/04 13:58
///ATTR SC,RW
///GROUP1 RB1,BS1
///GROUP2 ST1
NOP
'OK_r2_O38-47,64(2)(90,0)
'Down
MOVJ C00000 BC00000 VJ=100.00  +MOVJ EC00000 VJ=100.00
MOVJ C00001 BC00001 VJ=30.00  +MOVJ EC00001 VJ=100.00
'Path S1701
SFTOF3D
MOVJ C00002 BC00002 VJ=50.00  +MOVJ EC00002 VJ=100.00
MOVL C00003 BC00003 V=400.0  +MOVJ EC00003 VJ=100.00
SMOVL C00004 BC00004 V=100.0  +MOVJ EC00004
SREFP 3 C00005 BC00005  +REFP EC00005
CALL JOB:SEARCH-R1-S13D
SET P021 P006
SFTON3D P021
SMOVL C00006 BC00006 V=100.0  +MOVJ EC00006
SMOVL C00007 BC00007 V=100.0  +MOVJ EC00007
SMOVL C00008 BC00008 V=100.0  +MOVJ EC00008
SREFP 3 C00009 BC00009  +REFP EC00009
CALL JOB:SEARCH-R1-S13D
SET P021 P006
SFTON3D P021
SMOVL C00010 BC00010 V=100.0  +MOVJ EC00010
SMOVL C00011 BC00011 V=100.0  +MOVJ EC00011
MOVL C00012 BC00012 V=400.0  +MOVJ EC00012 VJ=100.00
MOVL C00013 BC00013 V=1000.0  +MOVJ EC00013 VJ=100.00
MOVJ C00014 BC00014 VJ=100.00  +MOVJ EC00014 VJ=100.00
MOVJ C00015 BC00015 VJ=100.00  +MOVJ EC00015 VJ=100.00
MOVJ C00016 BC00016 VJ=100.00  +MOVJ EC00016 VJ=100.00
MOVJ C00017 BC00017 VJ=100.00  +MOVJ EC00017 VJ=100.00
'Path S1702
SFTOF3D
MOVJ C00018 BC00018 VJ=100.00  +MOVJ EC00018 VJ=100.00
MOVL C00019 BC00019 V=166.7  +MOVJ EC00019 VJ=100.00
SMOVL C00020 BC00020 V=166.7  +MOVJ EC00020
SREFP 3 C00021 BC00021  +REFP EC00021
CALL JOB:SEARCH-R1-S13D
SET P022 P006
SFTON3D P022
SMOVL C00022 BC00022 V=100.0  +MOVJ EC00022
SMOVL C00023 BC00023 V=100.0  +MOVJ EC00023
SMOVL C00024 BC00024 V=100.0  +MOVJ EC00024
SREFP 3 C00025 BC00025  +REFP EC00025
CALL JOB:SEARCH-R1-S13D
SET P022 P006
SFTON3D P022
SMOVL C00026 BC00026 V=100.0  +MOVJ EC00026
SMOVL C00027 BC00027 V=250.0  +MOVJ EC00027
MOVL C00028 BC00028 V=1000.0  +MOVJ EC00028 VJ=100.00
MOVJ C00029 BC00029 VJ=100.00  +MOVJ EC00029 VJ=100.00
'Path S1703
SFTOF3D
MOVJ C00030 BC00030 VJ=100.00  +MOVJ EC00030 VJ=100.00
SMOVL C00031 BC00031 V=250.0  +MOVJ EC00031
SMOVL C00032 BC00032 V=100.0  +MOVJ EC00032
SREFP 3 C00033 BC00033  +REFP EC00033
CALL JOB:SEARCH-R1-S13D
SET P023 P006
SFTON3D P023
SMOVL C00034 BC00034 V=100.0  +MOVJ EC00034
SMOVL C00035 BC00035 V=100.0  +MOVJ EC00035
SREFP 3 C00036 BC00036  +REFP EC00036
CALL JOB:SEARCH-R1-S13D
SET P023 P006
SFTON3D P023
SMOVL C00037 BC00037 V=166.7  +MOVJ EC00037
MOVL C00038 BC00038 V=1000.0  +MOVJ EC00038 VJ=100.00
MOVL C00039 BC00039 V=1000.0  +MOVJ EC00039 VJ=100.00
MOVJ C00040 BC00040 VJ=100.00  +MOVJ EC00040 VJ=100.00
MOVJ C00041 BC00041 VJ=100.00  +MOVJ EC00041 VJ=100.00
MOVJ C00042 BC00042 VJ=100.00  +MOVJ EC00042 VJ=100.00
MOVJ C00043 BC00043 VJ=100.00  +MOVJ EC00043 VJ=100.00
MOVJ C00044 BC00044 VJ=100.00  +MOVJ EC00044 VJ=100.00
'Up
'Path S1246
SFTOF3D
MOVJ C00045 BC00045 VJ=100.00  +MOVJ EC00045 VJ=100.00
SMOVL C00046 BC00046 V=100.0  +MOVJ EC00046
SREFP 3 C00047 BC00047  +REFP EC00047
CALL JOB:SEARCH-R1-S13D
SET P030 P006
SFTON3D P030
SMOVL C00048 BC00048 V=100.0  +MOVJ EC00048
SREFP 3 C00049 BC00049  +REFP EC00049
CALL JOB:SEARCH-R1-S13D
SET P030 P006
SFTON3D P030
SMOVL C00050 BC00050 V=133.3  +MOVJ EC00050
SFTOF3D
MOVL C00051 BC00051 V=400.0  +MOVJ EC00051 VJ=100.00
SMOVL C00052 BC00052 V=100.0  +MOVJ EC00052
SREFP 3 C00053 BC00053  +REFP EC00053
CALL JOB:SEARCH-R1-S13D
SET P031 P006
SFTON3D P031
SMOVL C00054 BC00054 V=100.0  +MOVJ EC00054
SREFP 3 C00055 BC00055  +REFP EC00055
CALL JOB:SEARCH-R1-S13D
SET P031 P006
SFTON3D P031
SMOVL C00056 BC00056 V=133.3  +MOVJ EC00056
MOVL C00057 BC00057 V=1000.0  +MOVJ EC00057 VJ=100.00
'Path S1276
SFTOF3D
COMM PAUSE
COMM MOVJ C00058 BC00058 VJ=100.00  +MOVJ EC00058 VJ=100.00
COMM MOVL C00059 BC00059 V=400.0  +MOVJ EC00059 VJ=100.00
COMM SMOVL C00060 BC00060 V=100.0  +MOVJ EC00060
COMM SREFP 3 C00061 BC00061  +REFP EC00061
COMM CALL JOB:SEARCH-R1-S13D
COMM SET P032 P006
COMM SFTON3D P032
COMM SMOVL C00062 BC00062 V=100.0  +MOVJ EC00062
COMM SREFP 3 C00063 BC00063  +REFP EC00063
COMM CALL JOB:SEARCH-R1-S13D
COMM SET P032 P006
COMM SFTON3D P032
COMM SMOVL C00064 BC00064 V=100.0  +MOVJ EC00064
COMM MOVL C00065 BC00065 V=400.0  +MOVJ EC00065 VJ=100.00
COMM SFTOF3D
COMM MOVJ C00066 BC00066 VJ=100.00  +MOVJ EC00066 VJ=100.00
COMM SMOVL C00067 BC00067 V=100.0  +MOVJ EC00067
COMM SREFP 3 C00068 BC00068  +REFP EC00068
COMM CALL JOB:SEARCH-R1-S13D
COMM SET P033 P006
COMM SFTON3D P033
COMM SMOVL C00069 BC00069 V=100.0  +MOVJ EC00069
COMM SREFP 3 C00070 BC00070  +REFP EC00070
COMM CALL JOB:SEARCH-R1-S13D
COMM SET P033 P006
COMM SFTON3D P033
COMM SMOVL C00071 BC00071 V=100.0  +MOVJ EC00071
COMM SFTOF3D
COMM MOVL C00072 BC00072 V=400.0  +MOVJ EC00072 VJ=100.00
MOVJ C00073 BC00073 VJ=100.00  +MOVJ EC00073 VJ=100.00
SMOVL C00074 BC00074 V=100.0  +MOVJ EC00074
SREFP 3 C00075 BC00075  +REFP EC00075
CALL JOB:SEARCH-R1-S13D
SET P034 P006
SFTON3D P034
SMOVL C00076 BC00076 V=100.0  +MOVJ EC00076
SREFP 3 C00077 BC00077  +REFP EC00077
CALL JOB:SEARCH-R1-S13D
SET P034 P006
SFTON3D P034
SMOVL C00078 BC00078 V=100.0  +MOVJ EC00078
MOVL C00079 BC00079 V=400.0  +MOVJ EC00079 VJ=100.00
MOVJ C00080 BC00080 VJ=100.00  +MOVJ EC00080 VJ=100.00
'Path S1278
SFTOF3D
MOVJ C00081 BC00081 VJ=100.00  +MOVJ EC00081 VJ=100.00
SMOVL C00082 BC00082 V=100.0  +MOVJ EC00082
SREFP 3 C00083 BC00083  +REFP EC00083
CALL JOB:SEARCH-R1-S13D
SET P035 P006
SFTON3D P035
SMOVL C00084 BC00084 V=100.0  +MOVJ EC00084
SREFP 3 C00085 BC00085  +REFP EC00085
CALL JOB:SEARCH-R1-S13D
SET P035 P006
SFTON3D P035
SMOVL C00086 BC00086 V=100.0  +MOVJ EC00086
SFTOF3D
MOVL C00087 BC00087 V=400.0  +MOVJ EC00087 VJ=100.00
SMOVL C00088 BC00088 V=100.0  +MOVJ EC00088
SREFP 3 C00089 BC00089  +REFP EC00089
CALL JOB:SEARCH-R1-S13D
SET P036 P006
SFTON3D P036
SMOVL C00090 BC00090 V=100.0  +MOVJ EC00090
SREFP 3 C00091 BC00091  +REFP EC00091
CALL JOB:SEARCH-R1-S13D
SET P036 P006
SFTON3D P036
SMOVL C00092 BC00092 V=100.0  +MOVJ EC00092
'Path S1970
SFTOF3D
MOVJ C00093 BC00093 VJ=100.00  +MOVJ EC00093 VJ=100.00
MOVL C00094 BC00094 V=400.0  +MOVJ EC00094 VJ=100.00
SMOVL C00095 BC00095 V=100.0  +MOVJ EC00095
SREFP 3 C00096 BC00096  +REFP EC00096
CALL JOB:SEARCH-R1-S13D
SET P037 P006
SFTON3D P037
SMOVL C00097 BC00097 V=100.0  +MOVJ EC00097
SREFP 3 C00098 BC00098  +REFP EC00098
CALL JOB:SEARCH-R1-S13D
SET P037 P006
SFTON3D P037
SMOVL C00099 BC00099 V=100.0  +MOVJ EC00099
SFTOF3D
MOVL C00100 BC00100 V=400.0  +MOVJ EC00100 VJ=100.00
MOVL C00101 BC00101 V=1000.0  +MOVJ EC00101 VJ=100.00
COMM PAUSE
COMM MOVJ C00102 BC00102 VJ=100.00  +MOVJ EC00102 VJ=100.00
COMM SMOVL C00103 BC00103 V=100.0  +MOVJ EC00103
COMM SREFP 3 C00104 BC00104  +REFP EC00104
COMM CALL JOB:SEARCH-R1-S13D
COMM SET P038 P006
COMM SFTON3D P038
COMM SMOVL C00105 BC00105 V=100.0  +MOVJ EC00105
COMM SREFP 3 C00106 BC00106  +REFP EC00106
COMM CALL JOB:SEARCH-R1-S13D
COMM SET P038 P006
COMM SFTON3D P038
COMM SMOVL C00107 BC00107 V=100.0  +MOVJ EC00107
COMM SFTOF3D
COMM MOVL C00108 BC00108 V=400.0  +MOVJ EC00108 VJ=100.00
COMM SMOVL C00109 BC00109 V=100.0  +MOVJ EC00109
COMM SREFP 3 C00110 BC00110  +REFP EC00110
COMM CALL JOB:SEARCH-R1-S13D
COMM SET P039 P006
COMM SFTON3D P039
COMM SMOVL C00111 BC00111 V=100.0  +MOVJ EC00111
COMM SREFP 3 C00112 BC00112  +REFP EC00112
COMM CALL JOB:SEARCH-R1-S13D
COMM SET P039 P006
COMM SFTON3D P039
COMM SMOVL C00113 BC00113 V=100.0  +MOVJ EC00113
COMM MOVJ C00114 BC00114 VJ=100.00  +MOVJ EC00114 VJ=100.00
SFTOF3D
MOVJ C00115 BC00115 VJ=100.00  +MOVJ EC00115 VJ=100.00
MOVJ C00116 BC00116 VJ=100.00  +MOVJ EC00116 VJ=100.00
MOVJ C00117 BC00117 VJ=100.00  +MOVJ EC00117 VJ=100.00
MOVJ C00118 BC00118 VJ=100.00  +MOVJ EC00118 VJ=100.00
SMOVL C00119 BC00119 V=100.0  +MOVJ EC00119
SREFP 3 C00120 BC00120  +REFP EC00120
CALL JOB:SEARCH-R1-S13D
SET P040 P006
SFTON3D P040
SMOVL C00121 BC00121 V=100.0  +MOVJ EC00121
SREFP 3 C00122 BC00122  +REFP EC00122
CALL JOB:SEARCH-R1-S13D
SET P040 P006
SFTON3D P040
SMOVL C00123 BC00123 V=100.0  +MOVJ EC00123
SFTOF3D
MOVL C00124 BC00124 V=1000.0  +MOVJ EC00124 VJ=100.00
SMOVL C00125 BC00125 V=100.0  +MOVJ EC00125
SREFP 3 C00126 BC00126  +REFP EC00126
CALL JOB:SEARCH-R1-S13D
SET P041 P006
SFTON3D P041
SMOVL C00127 BC00127 V=100.0  +MOVJ EC00127
SREFP 3 C00128 BC00128  +REFP EC00128
CALL JOB:SEARCH-R1-S13D
SET P041 P006
SFTON3D P041
SMOVL C00129 BC00129 V=100.0  +MOVJ EC00129
MOVJ C00130 BC00130 VJ=100.00  +MOVJ EC00130 VJ=100.00
SFTOF3D
MOVJ C00131 BC00131 VJ=100.00  +MOVJ EC00131 VJ=100.00
MOVL C00132 BC00132 V=400.0  +MOVJ EC00132 VJ=100.00
SMOVL C00133 BC00133 V=100.0  +MOVJ EC00133
SREFP 3 C00134 BC00134  +REFP EC00134
CALL JOB:SEARCH-R1-S13D
SET P042 P006
SFTON3D P042
SMOVL C00135 BC00135 V=100.0  +MOVJ EC00135
SREFP 3 C00136 BC00136  +REFP EC00136
CALL JOB:SEARCH-R1-S13D
SET P042 P006
SFTON3D P042
SMOVL C00137 BC00137 V=100.0  +MOVJ EC00137
SFTOF3D
MOVL C00138 BC00138 V=400.0  +MOVJ EC00138 VJ=100.00
'Path S1282
SFTOF3D
SMOVL C00139 BC00139 V=100.0  +MOVJ EC00139
SREFP 3 C00140 BC00140  +REFP EC00140
CALL JOB:SEARCH-R1-S13D
SET P043 P006
SFTON3D P043
SMOVL C00141 BC00141 V=100.0  +MOVJ EC00141
SREFP 3 C00142 BC00142  +REFP EC00142
CALL JOB:SEARCH-R1-S13D
SET P043 P006
SFTON3D P043
SMOVL C00143 BC00143 V=100.0  +MOVJ EC00143
SFTOF3D
MOVL C00144 BC00144 V=400.0  +MOVJ EC00144 VJ=100.00
MOVL C00145 BC00145 V=1000.0  +MOVJ EC00145 VJ=100.00
MOVJ C00146 BC00146 VJ=100.00  +MOVJ EC00146 VJ=100.00
MOVJ C00147 BC00147 VJ=100.00  +MOVJ EC00147 VJ=100.00
MOVL C00148 BC00148 V=400.0  +MOVJ EC00148 VJ=100.00
SMOVL C00149 BC00149 V=100.0  +MOVJ EC00149
SREFP 3 C00150 BC00150  +REFP EC00150
CALL JOB:SEARCH-R1-S13D
SET P044 P006
SFTON3D P044
SMOVL C00151 BC00151 V=100.0  +MOVJ EC00151
SREFP 3 C00152 BC00152  +REFP EC00152
CALL JOB:SEARCH-R1-S13D
SET P044 P006
SFTON3D P044
SMOVL C00153 BC00153 V=100.0  +MOVJ EC00153
MOVL C00154 BC00154 V=400.0  +MOVJ EC00154 VJ=100.00
SFTON3D P044
SMOVL C00155 BC00155 V=133.3 PL=0  +MOVJ EC00155
SREFP 1 C00156 BC00156  +REFP EC00156
SREFP 2 C00157 BC00157  +REFP EC00157
MACRO1 MJ#(0) ARGF9
ARCON
SWVON WEV#(60)
SMOVL C00158 BC00158 V=8.3  +MOVJ EC00158
SMOVL C00159 BC00159 V=8.3  +MOVJ EC00159
SMOVL C00160 BC00160 V=8.3  +MOVJ EC00160
ARCOF
SWVOF
SMOVL C00161 BC00161 V=250.0  +MOVJ EC00161
SFTOF3D
MOVJ C00162 BC00162 VJ=100.00  +MOVJ EC00162 VJ=100.00
SFTOF3D
MOVJ C00163 BC00163 VJ=70.00  +MOVJ EC00163 VJ=100.00
'Path W1138
MOVJ C00164 BC00164 VJ=100.00  +MOVJ EC00164 VJ=100.00
SFTOF
SFTON3D P037
SMOVL C00165 BC00165 V=133.3 PL=0  +MOVJ EC00165
SREFP 1 C00166 BC00166  +REFP EC00166
SREFP 2 C00167 BC00167  +REFP EC00167
MACRO1 MJ#(0) ARGF9
ARCON
SWVON WEV#(60)
SMOVL C00168 BC00168 V=8.3  +MOVJ EC00168
SMOVL C00169 BC00169 V=8.3  +MOVJ EC00169
SMOVL C00170 BC00170 V=8.3  +MOVJ EC00170
ARCOF
SWVOF
SMOVL C00171 BC00171 V=400.0  +MOVJ EC00171
MOVJ C00172 BC00172 VJ=100.00  +MOVJ EC00172 VJ=100.00
SFTOF3D
COMM PAUSE
COMM MOVJ C00173 BC00173 VJ=100.00  +MOVJ EC00173 VJ=100.00
COMM MOVJ C00174 BC00174 VJ=100.00  +MOVJ EC00174 VJ=100.00
COMM SFTON3D P039
COMM SMOVL C00175 BC00175 V=133.3 PL=0  +MOVJ EC00175
COMM SREFP 1 C00176 BC00176  +REFP EC00176
COMM SREFP 2 C00177 BC00177  +REFP EC00177
COMM MACRO1 MJ#(0) ARGF14
COMM ARCON
COMM SFTON3D P038
COMM SMOVL C00178 BC00178 V=8.3  +MOVJ EC00178
COMM SMOVL C00179 BC00179 V=8.3  +MOVJ EC00179
COMM ARCOF
COMM SMOVL C00180 BC00180 V=400.0  +MOVJ EC00180
COMM SFTOF3D
COMM MOVJ C00181 BC00181 VJ=100.00  +MOVJ EC00181 VJ=100.00
COMM MOVJ C00182 BC00182 VJ=100.00  +MOVJ EC00182 VJ=100.00
COMM MOVJ C00183 BC00183 VJ=100.00  +MOVJ EC00183 VJ=100.00
COMM MOVJ C00184 BC00184 VJ=100.00  +MOVJ EC00184 VJ=100.00
COMM 'Path W1140
COMM SFTOF3D
COMM SFTON3D P033
COMM SMOVL C00185 BC00185 V=133.3 PL=0  +MOVJ EC00185
COMM SREFP 1 C00186 BC00186  +REFP EC00186
COMM SREFP 2 C00187 BC00187  +REFP EC00187
COMM MACRO1 MJ#(0) ARGF14
COMM ARCON
COMM SWVON WEV#(10)
COMM SMOVL C00188 BC00188 V=8.3  +MOVJ EC00188
COMM SFTON3D P032
COMM SMOVL C00189 BC00189 V=8.3  +MOVJ EC00189
COMM SMOVL C00190 BC00190 V=8.3  +MOVJ EC00190
COMM ARCOF
COMM SWVOF
COMM SMOVL C00191 BC00191 V=400.0  +MOVJ EC00191
COMM SFTOF3D
COMM MOVJ C00192 BC00192 VJ=100.00  +MOVJ EC00192 VJ=100.00
SFTOF3D
MOVJ C00193 BC00193 VJ=100.00  +MOVJ EC00193 VJ=100.00
'Path W1142
SFTOF3D
SFTON3D P030
MOVJ C00194 BC00194 VJ=100.00  +MOVJ EC00194 VJ=100.00
SMOVL C00195 BC00195 V=133.3 PL=0  +MOVJ EC00195
SREFP 1 C00196 BC00196  +REFP EC00196
SREFP 2 C00197 BC00197  +REFP EC00197
MACRO1 MJ#(0) ARGF9
ARCON
SMOVL C00198 BC00198 V=8.3  +MOVJ EC00198
SFTON3D P031
SMOVL C00199 BC00199 V=8.3  +MOVJ EC00199
SMOVL C00200 BC00200 V=8.3  +MOVJ EC00200
SMOVL C00201 BC00201 V=8.3  +MOVJ EC00201
ARCOF
SMOVL C00202 BC00202 V=400.0  +MOVJ EC00202
SFTOF3D
MOVJ C00203 BC00203 VJ=100.00  +MOVJ EC00203 VJ=100.00
'Path W1143
SFTOF3D
SFTON3D P034
MOVJ C00204 BC00204 VJ=100.00  +MOVJ EC00204 VJ=100.00
SMOVL C00205 BC00205 V=133.3 PL=0  +MOVJ EC00205
SREFP 1 C00206 BC00206  +REFP EC00206
SREFP 2 C00207 BC00207  +REFP EC00207
MACRO1 MJ#(0) ARGF9
ARCON
SMOVC C00208 BC00208 V=8.3  +MOVJ EC00208
SMOVC C00209 BC00209 V=8.3  +MOVJ EC00209
SMOVC C00210 BC00210 V=8.3  +MOVJ EC00210
SMOVL C00211 BC00211 V=8.3  +MOVJ EC00211
SMOVC C00212 BC00212 V=8.3  +MOVJ EC00212
SMOVC C00213 BC00213 V=8.3  +MOVJ EC00213
SMOVC C00214 BC00214 V=8.3  +MOVJ EC00214
ARCOF
SMOVL C00215 BC00215 V=400.0  +MOVJ EC00215
SFTOF3D
MOVJ C00216 BC00216 VJ=100.00  +MOVJ EC00216 VJ=100.00
'Path W1144
SFTOF3D
SFTON3D P036
MOVJ C00217 BC00217 VJ=100.00  +MOVJ EC00217 VJ=100.00
SFTON3D P036
SMOVL C00218 BC00218 V=133.3 PL=0  +MOVJ EC00218
SREFP 1 C00219 BC00219  +REFP EC00219
SREFP 2 C00220 BC00220  +REFP EC00220
MACRO1 MJ#(0) ARGF14
ARCON
SMOVL C00221 BC00221 V=9.2  +MOVJ EC00221
SFTON3D P035
SMOVL C00222 BC00222 V=9.2  +MOVJ EC00222
SMOVL C00223 BC00223 V=9.2  +MOVJ EC00223
ARCOF
SMOVL C00224 BC00224 V=400.0  +MOVJ EC00224
SFTOF3D
MOVJ C00225 BC00225 VJ=100.00  +MOVJ EC00225 VJ=100.00
MOVJ C00226 BC00226 VJ=100.00  +MOVJ EC00226 VJ=100.00
SFTON3D P042
SMOVL C00227 BC00227 V=133.3 PL=0  +MOVJ EC00227
SREFP 1 C00228 BC00228  +REFP EC00228
SREFP 2 C00229 BC00229  +REFP EC00229
MACRO1 MJ#(0) ARGF14
ARCON
SMOVL C00230 BC00230 V=10.0  +MOVJ EC00230
SFTON3D P043
SMOVL C00231 BC00231 V=10.0  +MOVJ EC00231
SMOVL C00232 BC00232 V=10.0  +MOVJ EC00232
ARCOF
SMOVL C00233 BC00233 V=400.0  +MOVJ EC00233
MOVJ C00234 BC00234 VJ=100.00  +MOVJ EC00234 VJ=100.00
MOVJ C00235 BC00235 VJ=100.00  +MOVJ EC00235 VJ=100.00
SFTOF3D
SFTON3D P040
SMOVL C00236 BC00236 V=133.3 PL=0  +MOVJ EC00236
SREFP 1 C00237 BC00237  +REFP EC00237
SREFP 2 C00238 BC00238  +REFP EC00238
MACRO1 MJ#(0) ARGF14
ARCON
SMOVL C00239 BC00239 V=10.0  +MOVJ EC00239
SFTON3D P041
SMOVL C00240 BC00240 V=10.0  +MOVJ EC00240
SMOVL C00241 BC00241 V=10.0  +MOVJ EC00241
ARCOF
SMOVL C00242 BC00242 V=400.0  +MOVJ EC00242
SFTOF3D
MOVJ C00243 BC00243 VJ=100.00  +MOVJ EC00243 VJ=100.00
MOVJ C00244 BC00244 VJ=100.00  +MOVJ EC00244 VJ=100.00
MOVJ C00245 BC00245 VJ=100.00  +MOVJ EC00245 VJ=100.00
MOVJ C00246 BC00246 VJ=100.00  +MOVJ EC00246 VJ=100.00
MOVJ C00247 BC00247 VJ=100.00  +MOVJ EC00247 VJ=100.00
'Down
'1
MOVJ C00248 BC00248 VJ=100.00  +MOVJ EC00248 VJ=100.00
'Path W1705
SFTOF3D
SFTON3D P023
MOVJ C00249 BC00249 VJ=100.00  +MOVJ EC00249 VJ=100.00
SMOVL C00250 BC00250 V=400.0  +MOVJ EC00250
SMOVL C00251 BC00251 V=133.3 PL=0  +MOVJ EC00251
SREFP 1 C00252 BC00252  +REFP EC00252
SREFP 2 C00253 BC00253  +REFP EC00253
MACRO1 MJ#(0) ARGF14
ARCON
SMOVL C00254 BC00254 V=10.0  +MOVJ EC00254
SMOVL C00255 BC00255 V=10.0  +MOVJ EC00255
SMOVL C00256 BC00256 V=10.0  +MOVJ EC00256
ARCOF
SMOVL C00257 BC00257 V=400.0  +MOVJ EC00257
SMOVL C00258 BC00258 V=1000.0  +MOVJ EC00258
SFTOF3D
MOVJ C00259 BC00259 VJ=100.00  +MOVJ EC00259 VJ=100.00
MOVJ C00260 BC00260 VJ=100.00  +MOVJ EC00260 VJ=100.00
'2
MOVJ C00261 BC00261 VJ=100.00  +MOVJ EC00261 VJ=100.00
MOVJ C00262 BC00262 VJ=100.00  +MOVJ EC00262 VJ=100.00
MOVJ C00263 BC00263 VJ=100.00  +MOVJ EC00263 VJ=100.00
'Path W1706
SFTOF3D
SFTON3D P021
MOVJ C00264 BC00264 VJ=15.00  +MOVJ EC00264 VJ=100.00
SMOVL C00265 BC00265 V=400.0  +MOVJ EC00265
SMOVL C00266 BC00266 V=100.0 PL=0  +MOVJ EC00266
SREFP 1 C00267 BC00267  +REFP EC00267
SREFP 2 C00268 BC00268  +REFP EC00268
MACRO1 MJ#(0) ARGF14
ARCON
SMOVL C00269 BC00269 V=10.0  +MOVJ EC00269
ARCOF
SMOVL C00270 BC00270 V=400.0  +MOVJ EC00270
SMOVL C00271 BC00271 V=1000.0  +MOVJ EC00271
SFTOF3D
MOVJ C00272 BC00272 VJ=50.00  +MOVJ EC00272 VJ=100.00
'Path W1707
SFTOF3D
SFTON3D P021
MOVJ C00273 BC00273 VJ=100.00  +MOVJ EC00273 VJ=100.00
SMOVL C00274 BC00274 V=400.0  +MOVJ EC00274
SMOVL C00275 BC00275 V=100.0 PL=0  +MOVJ EC00275
SREFP 1 C00276 BC00276  +REFP EC00276
SREFP 2 C00277 BC00277  +REFP EC00277
MACRO1 MJ#(0) ARGF14
ARCON
SMOVL C00278 BC00278 V=10.0  +MOVJ EC00278
ARCOF
SMOVL C00279 BC00279 V=400.0  +MOVJ EC00279
SMOVL C00280 BC00280 V=1000.0  +MOVJ EC00280
SFTOF3D
MOVJ C00281 BC00281 VJ=100.00  +MOVJ EC00281 VJ=100.00
MOVJ C00282 BC00282 VJ=100.00  +MOVJ EC00282 VJ=100.00
'3
MOVJ C00283 BC00283 VJ=100.00  +MOVJ EC00283 VJ=100.00
MOVJ C00284 BC00284 VJ=100.00  +MOVJ EC00284 VJ=100.00
'Path W1709
SFTOF3D
SFTON3D P023
MOVJ C00285 BC00285 VJ=100.00  +MOVJ EC00285 VJ=100.00
SMOVL C00286 BC00286 V=400.0  +MOVJ EC00286
SMOVL C00287 BC00287 V=133.3 PL=0  +MOVJ EC00287
SREFP 1 C00288 BC00288  +REFP EC00288
SREFP 2 C00289 BC00289  +REFP EC00289
MACRO1 MJ#(0) ARGF14
ARCON
SMOVL C00290 BC00290 V=10.0  +MOVJ EC00290
SMOVL C00291 BC00291 V=10.0  +MOVJ EC00291
SMOVL C00292 BC00292 V=10.0  +MOVJ EC00292
ARCOF
SMOVL C00293 BC00293 V=400.0  +MOVJ EC00293
SMOVL C00294 BC00294 V=1000.0  +MOVJ EC00294
SFTOF3D
MOVJ C00295 BC00295 VJ=100.00  +MOVJ EC00295 VJ=100.00
MOVJ C00296 BC00296 VJ=100.00  +MOVJ EC00296 VJ=100.00
'4
MOVJ C00297 BC00297 VJ=100.00  +MOVJ EC00297 VJ=100.00
MOVJ C00298 BC00298 VJ=100.00  +MOVJ EC00298 VJ=100.00
'Path W1710
SFTOF3D
SFTON3D P021
MOVJ C00299 BC00299 VJ=15.00  +MOVJ EC00299 VJ=100.00
SMOVL C00300 BC00300 V=400.0  +MOVJ EC00300
SMOVL C00301 BC00301 V=133.3 PL=0  +MOVJ EC00301
SREFP 1 C00302 BC00302  +REFP EC00302
SREFP 2 C00303 BC00303  +REFP EC00303
MACRO1 MJ#(0) ARGF14
ARCON
SMOVL C00304 BC00304 V=10.0  +MOVJ EC00304
ARCOF
SMOVL C00305 BC00305 V=400.0  +MOVJ EC00305
SMOVL C00306 BC00306 V=1000.0  +MOVJ EC00306
SFTOF3D
'Path W1711
SFTOF3D
SFTON3D P021
MOVJ C00307 BC00307 VJ=100.00  +MOVJ EC00307 VJ=100.00
SMOVL C00308 BC00308 V=400.0  +MOVJ EC00308
SMOVL C00309 BC00309 V=133.3 PL=0  +MOVJ EC00309
SREFP 1 C00310 BC00310  +REFP EC00310
SREFP 2 C00311 BC00311  +REFP EC00311
MACRO1 MJ#(0) ARGF14
ARCON
SMOVL C00312 BC00312 V=10.0  +MOVJ EC00312
ARCOF
SMOVL C00313 BC00313 V=400.0  +MOVJ EC00313
SMOVL C00314 BC00314 V=1000.0  +MOVJ EC00314
SFTOF3D
MOVJ C00315 BC00315 VJ=100.00  +MOVJ EC00315 VJ=100.00
MOVJ C00316 BC00316 VJ=100.00  +MOVJ EC00316 VJ=100.00
'6
MOVJ C00317 BC00317 VJ=100.00  +MOVJ EC00317 VJ=100.00
MOVJ C00318 BC00318 VJ=100.00  +MOVJ EC00318 VJ=100.00
'Path W1714
SFTOF3D
SFTON3D P022
MOVJ C00319 BC00319 VJ=100.00  +MOVJ EC00319 VJ=100.00
SMOVL C00320 BC00320 V=400.0  +MOVJ EC00320
SMOVL C00321 BC00321 V=133.3 PL=0  +MOVJ EC00321
SREFP 1 C00322 BC00322  +REFP EC00322
SREFP 2 C00323 BC00323  +REFP EC00323
MACRO1 MJ#(0) ARGF14
ARCON
SMOVL C00324 BC00324 V=10.0  +MOVJ EC00324
ARCOF
SMOVL C00325 BC00325 V=400.0  +MOVJ EC00325
SMOVL C00326 BC00326 V=1000.0  +MOVJ EC00326
SFTOF3D
'Path W1715
SFTOF3D
SFTON3D P022
MOVJ C00327 BC00327 VJ=100.00  +MOVJ EC00327 VJ=100.00
SMOVL C00328 BC00328 V=400.0  +MOVJ EC00328
SMOVL C00329 BC00329 V=133.3 PL=0  +MOVJ EC00329
SREFP 1 C00330 BC00330  +REFP EC00330
SREFP 2 C00331 BC00331  +REFP EC00331
MACRO1 MJ#(0) ARGF14
ARCON
SMOVL C00332 BC00332 V=10.0  +MOVJ EC00332
ARCOF
SMOVL C00333 BC00333 V=400.0  +MOVJ EC00333
SFTOF3D
MOVJ C00334 BC00334 VJ=100.00  +MOVJ EC00334 VJ=14.00
MOVJ C00335 BC00335 VJ=100.00  +MOVJ EC00335 VJ=100.00
MOVJ C00336 BC00336 VJ=100.00  +MOVJ EC00336 VJ=100.00
MOVJ C00337 BC00337 VJ=100.00  +MOVJ EC00337 VJ=100.00
MOVJ C00338 BC00338 VJ=100.00  +MOVJ EC00338 VJ=100.00
'7
MOVJ C00339 BC00339 VJ=100.00  +MOVJ EC00339 VJ=100.00
'Path W1716
SFTOF3D
SFTON3D P022
MOVJ C00340 BC00340 VJ=100.00  +MOVJ EC00340 VJ=25.00
MOVJ C00341 BC00341 VJ=100.00  +MOVJ EC00341 VJ=100.00
SMOVL C00342 BC00342 V=400.0  +MOVJ EC00342
SMOVL C00343 BC00343 V=133.3 PL=0  +MOVJ EC00343
SREFP 1 C00344 BC00344  +REFP EC00344
SREFP 2 C00345 BC00345  +REFP EC00345
MACRO1 MJ#(0) ARGF14
ARCON
SMOVL C00346 BC00346 V=11.7  +MOVJ EC00346
ARCOF
SMOVL C00347 BC00347 V=400.0  +MOVJ EC00347
SFTOF3D
MOVJ C00348 BC00348 VJ=50.00  +MOVJ EC00348 VJ=100.00
MOVJ C00349 BC00349 VJ=100.00  +MOVJ EC00349 VJ=25.00
MOVJ C00350 BC00350 VJ=30.00  +MOVJ EC00350 VJ=100.00
'Path W1717
SFTOF3D
SFTON3D P022
MOVJ C00351 BC00351 VJ=30.00  +MOVJ EC00351 VJ=100.00
SMOVL C00352 BC00352 V=400.0  +MOVJ EC00352
SMOVL C00353 BC00353 V=133.3 PL=0  +MOVJ EC00353
SREFP 1 C00354 BC00354  +REFP EC00354
SREFP 2 C00355 BC00355  +REFP EC00355
MACRO1 MJ#(0) ARGF14
ARCON
SMOVL C00356 BC00356 V=11.7  +MOVJ EC00356
ARCOF
SMOVL C00357 BC00357 V=400.0  +MOVJ EC00357
SMOVL C00358 BC00358 V=1000.0  +MOVJ EC00358
SFTOF3D
END
